// TIA Portal V17 export
// export: Created 2025-03-07T09:18:29.8996951Z, ExportSetting WithDefaults, DisplayName Totally Integrated Automation Portal, DisplayVersion V17 Update 8, DisplayName TIA Portal Openness, DisplayVersion V17 Update 8, DisplayName TIA Portal Version Control Interface, DisplayVersion V17, DisplayName SINAMICS Startdrive Advanced, DisplayVersion V17 SP2, DisplayName SINAMICS Startdrive G110M, G120, G120C, G120D, G120P, G115D, DisplayVersion V17 SP2, DisplayName SINAMICS Startdrive G130, G150, S120, S150, SINAMICS MV, S210, DisplayVersion V17 SP2, DisplayName STEP 7 Professional, DisplayVersion V17 Update 8, DisplayName SINUMERIK ONE STEP 7 Toolbox, DisplayVersion V17 Update 12, DisplayName SINUMERIK 840D sl STEP 7 Toolbox, DisplayVersion V17 Update 12, DisplayName STEP 7 Safety, DisplayVersion V17 Update 6, DisplayName WinCC Advanced, DisplayVersion V17 Update 8
DATA_BLOCK "LTLP_CycleTimeDB"   // DB523
{ DB_Accessible_From_OPC_UA := 'FALSE' }
// stored: AutoNumber true, DBAccessibleFromOPCUA false, DBAccessibleFromWebserver true, InstanceOfName LTLP_CycleTime, InstanceOfType FB
"LTLP_CycleTime"
   // VAR_INPUT
   //    MACHINING_UNIT : Int;
   //    RESTART_PLC : Bool;
   //    START : Bool;
   //    STOP : Bool;
   //    START_STOP : Bool;
   //    HOLD : Bool;
   // END_VAR
   // VAR_OUTPUT
   //    ERROR : Word;
   // END_VAR
   // VAR_IN_OUT
   //    HMI_DB : "LTLP_typeHmiProInterface";
   // END_VAR
   // VAR
   //    stationData : Array[0..40] of Struct
   //       trigger : Struct
   //          p_start : Bool;
   //          p_stop : Bool;
   //          p_hold : Bool;
   //          n_hold : Bool;
   //          p_start_stop : Bool;
   //          n_start_stop : Bool;
   //          res06 : Bool;
   //          res07 : Bool;
   //       END_STRUCT;
   //       impulse : Struct
   //          p_start : Bool;
   //          p_stop : Bool;
   //          p_hold : Bool;
   //          n_hold : Bool;
   //          p_start_stop : Bool;
   //          n_start_stop : Bool;
   //          res26 : Bool;
   //          res27 : Bool;
   //       END_STRUCT;
   //       mode : Struct
   //          shs_on : Bool;
   //          ss_on : Bool;
   //          res42 : Bool;
   //          res43 : Bool;
   //          res44 : Bool;
   //          res45 : Bool;
   //          res46 : Bool;
   //          res47 : Bool;
   //       END_STRUCT;
   //       StartTime : Time;
   //       SaveTime : Time;
   //       DiffTime : Time;
   //    END_STRUCT;
   //    fpRestartPLC : Bool;
   // END_VAR
BEGIN
END_DATA_BLOCK
